// Mitsubishi GX Works2 project: 수위제어풀이1   PLC: Q02/Q02H

PROGRAM MAIN
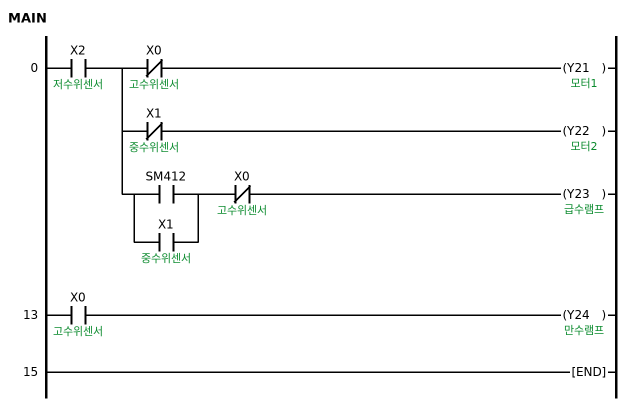
0     LD      X2  ; 저수위센서
      MPS
      ANI     X0  ; 고수위센서
      OUT     Y21  ; 모터1
      MRD
      ANI     X1  ; 중수위센서
      OUT     Y22  ; 모터2
      MPP
      LD      SM412
      OR      X1  ; 중수위센서
      ANB
      ANI     X0  ; 고수위센서
      OUT     Y23  ; 급수램프
13    LD      X0  ; 고수위센서
      OUT     Y24  ; 만수램프
15    END
END_PROGRAM

// device comments not shown above
M0  ; 보조0
M1  ; 보조1
M2  ; 보조2
M3  ; 보조3
